// TwinCAT 3 PLC project PLC1
// ProgramVersion: 3.1.4026.22
// libraries:
//   Tc2_EtherCAT, * (Beckhoff Automation GmbH)
//   Tc2_Standard, * (Beckhoff Automation GmbH)
//   Tc2_System, * (Beckhoff Automation GmbH)
//   Tc3_RealtimeMonitoring, * (Beckhoff Automation GmbH)
// project tree:
//   GVL/ FB_DoWork.TcPOU, GVL.TcGVL
//   POUs/ F_ConsumeTime.TcPOU, PRG_Task1.TcPOU, PRG_Task2.TcPOU, PRG_Task3.TcPOU
//   / Task1.TcTTO, Task2.TcTTO, Task3.TcTTO
// real-time tasks:
//   TASK Plc1Task: cycle T#10ms, priority 20, ADS port 350
//   TASK Plc2Task: cycle T#10ms, priority 21, ADS port 351
//   TASK ProviderPLC: cycle T#10ms, priority 13, ADS port 352

CONFIGURATION PLC1
    RESOURCE PLC ON TwinCAT3
        TASK Task1(INTERVAL := T#10ms, PRIORITY := 20);
        TASK Task2(INTERVAL := T#10ms, PRIORITY := 21);
        TASK Task3(INTERVAL := T#10ms, PRIORITY := 13);
        PROGRAM PRG_Task1 WITH Task1 : PRG_Task1;
        PROGRAM PRG_Task2 WITH Task2 : PRG_Task2;
        PROGRAM PRG_Task3 WITH Task3 : PRG_Task3;
    END_RESOURCE
END_CONFIGURATION

// ---- GVL/GVL.TcGVL
{attribute 'qualified_only'}
VAR_GLOBAL
	fbCrititcalSection : FB_IecCriticalSection;
	fbDoWork		   : FB_DoWork;
END_VAR

// ---- POUs/PRG_Task1.TcPOU
PROGRAM PRG_Task1
VAR
	{attribute 'displaymode':='hex'} 
	CallingTaskAdsPort :UINT;
END_VAR
VAR CONSTANT
//10 Microseconds gives enough time to ensure that Task 3 calls
//GVL.fbDoWork.M_Increment method before Task1.	
	DelayToCallInterface : UDINT := 10; 	
END_VAR

F_ConsumeTime(DelayToCallInterface);

CallingTaskAdsPort:=_TaskInfo[GETCURTASKINDEXEX()].AdsPort;

IF GVL.fbCrititcalSection.Enter() THEN
	(* start of critical section *)
	GVL.fbDoWork.M_ConsumeTime(CallerTaskAdsPort :=CallingTaskAdsPort );

	(* end of critical section *)
	GVL.fbCrititcalSection.Leave();
END_IF

END_PROGRAM

// ---- POUs/F_ConsumeTime.TcPOU
FUNCTION F_ConsumeTime
VAR_INPUT
	Us		:UDINT;
END_VAR
VAR
		tCurr, tEnd : T_DCTIME64;
END_VAR

tCurr := F_GetActualDcTime64();
tEnd  := tCurr + (Us * EC_DCTIME_TICKSPERMSEC64 / 1000);
WHILE (tCurr < tEnd) DO
	tCurr := F_GetActualDcTime64();
END_WHILE

END_FUNCTION

// ---- POUs/PRG_Task2.TcPOU
PROGRAM PRG_Task2
VAR
	//Just another task on the same core as task 1 to show the
	//scedular executing another task while task 1 gets blocked
END_VAR

F_ConsumeTime(400);

END_PROGRAM

// ---- POUs/PRG_Task3.TcPOU
PROGRAM PRG_Task3
VAR
	{attribute 'displaymode':='hex'} 
	CallingTaskAdsPort :UINT;	
END_VAR

CallingTaskAdsPort:=_TaskInfo[GETCURTASKINDEXEX()].AdsPort;

IF GVL.fbCrititcalSection.Enter() THEN
	(* start of critical section *)
	GVL.fbDoWork.M_ConsumeTime(CallerTaskAdsPort :=CallingTaskAdsPort );

	(* end of critical section *)
	GVL.fbCrititcalSection.Leave();
END_IF

END_PROGRAM

// ---- GVL/FB_DoWork.TcPOU
FUNCTION_BLOCK FB_DoWork

METHOD M_ConsumeTime : Global.HRESULT
VAR_INPUT
	CallerTaskAdsPort : UINT;
END_VAR

VAR_INST
	fbRTMon_LogMark : FB_RTMon_LogMark;
END_VAR
fbRTMon_LogMark.LogStart(CallerTaskAdsPort, 0);
F_ConsumeTime(100);
fbRTMon_LogMark.LogStop(CallerTaskAdsPort, 0);
END_METHOD

END_FUNCTION_BLOCK
